(* PLC project Generated.project, CODESYS CODESYS V3.5 SP19 Patch 1 *)
(* stored: creationDateTime 2026-09-03T04:58:03.489479, modificationDateTime 2026-09-03T04:58:03.489479 *)

(* values of E_CycleStep: X0_PREPARATION: Début de graphe : à la TRÉMIE, treuils en position HAUTE; X1_HOMING: Vitesses lentes pour chercher capteur top + référencement; X2_WORK_POS_SELECT: Sélection cible Trémie/P1/Maintenance + translation validée; X3_OPEN_BUCKET: Ouverture benne (si déjà ouverte -> passe vite); X4_DESCEND_OPEN: Plongée benne ouverte, M1+M2 synchro, Kobold mesure ON; X5_BOTTOM_CONFIRMED: Fond validé (FB_DiveSearch) ; arrêt descente; X6_CLOSE_BUCKET: Fermeture benne — tolérance « à peu près fermé »; X7_CTRL_ASCENT: Remontée palier 1 de contrôle; X8_ASCENT_LOADED: Remontée nominale jusqu'à limite haute; X9_DRAIN_PAUSE: Égouttage temporisé — durée configurable / passable IHM; X10_TRANSLATE_DUMP: Translation vers trémie (départ P1) + avertissements IHM; X11A_DUMP_ARRIVE: Arrivée trémie : treuils à l'arrêt, attente geste opérateur (ex-X11); X13_DONE_SYNC: Fin de cycle, synchronisation finale (R4) + compteur + durée cycle; STABILIZING: État d'attente/stabilisation — pas une erreur; X11B_DUMP_OPEN: Vidage à la trémie : ouverture benne, LES DEUX treuils à l'arrêt (aucune descente couplée); X11C_DUMP_REPOSITION: Repositionnement couplé M1+M2 (option IHM maintenue) : descente lente pour dégager la vidange, retour X11b au relâchement *)

{attribute 'qualified_only'}
{attribute 'strict'}
TYPE E_CycleStep : (X0_PREPARATION := 0, X1_HOMING := 1, X2_WORK_POS_SELECT := 2, X3_OPEN_BUCKET := 3, X4_DESCEND_OPEN := 4, X5_BOTTOM_CONFIRMED := 5, X6_CLOSE_BUCKET := 6, X7_CTRL_ASCENT := 7, X8_ASCENT_LOADED := 8, X9_DRAIN_PAUSE := 9, X10_TRANSLATE_DUMP := 10, X11A_DUMP_ARRIVE := 11, X13_DONE_SYNC := 13, STABILIZING := 14, X11B_DUMP_OPEN := 15, X11C_DUMP_REPOSITION := 16);
END_TYPE
